// TIA Portal project "MPS_4S_V13_SP1" (V13)

(* hardware
DEVICE "S7300/ET200M-Station_1"  S7-300 station
   slot 0: "Profilschiene_0"  Rail  6ES7 390-1***0-0AA0
   slot 1: "PS 307 5A_1"  PS 307 5A  6ES7 307-1EA00-0AA0
   slot 2: "S7-300 PLC"  CPU 314C-2 PN/DP  6ES7 314-6EH04-0AB0  V3.3
      slot 2: "PROFINET-Schnittstelle_1"  PN-IO
         slot 1: "Port_1"  Port
         slot 2: "Port_2"  Port
      slot 5: "DI 24/DO 16_1"  DI24/DO16
      slot 6: "AI 5/AO 2_1"  AI5/AO2
      slot 7: "Zählen_1"  Counter
      slot 8: "Positionieren_1"  Positioning
   slot 4: "CP 343-2_1"  CP 343-2  6GK7 343-2AH01-0XA0  V3.1
DEVICE "MPS Verteilen"  ET 200S station
   slot 0: "Baugruppenträger_0"  Rail
   slot 0: "Verteilen"  IM 151-1 Standard  6ES7 151-1AA04-0AB0
   slot 1: "PM-E DC24V_1"  PM-E 24VDC  6ES7 138-4CA01-0AA0
   slot 2: "4DI x DC24V ST_1"  4DI x 24VDC ST  6ES7 131-4BD01-0AA0
   slot 3: "4DI x DC24V ST_2"  4DI x 24VDC ST  6ES7 131-4BD01-0AA0
   slot 4: "4DO x DC24V / 0,5A ST_1"  4DO x 24VDC / 0.5A ST  6ES7 132-4BD02-0AA0
   slot 5: "4DO x DC24V / 0,5A ST_2"  4DO x 24VDC / 0.5A ST  6ES7 132-4BD02-0AA0
   slot 6: "4DI x DC24V ST_3"  4DI x 24VDC ST  6ES7 131-4BD01-0AA0
   slot 7: "4DO x DC24V / 0,5A ST_3"  4DO x 24VDC / 0.5A ST  6ES7 132-4BD02-0AA0
   slot 8: "4DO x DC24V / 0,5A ST_4"  4DO x 24VDC / 0.5A ST  6ES7 132-4BD02-0AA0
DEVICE "MPS Pick and Place"  ET 200S station
   slot 0: "Baugruppenträger_0"  Rail
   slot 0: "Pick and Place"  IM 151-1 Standard  6ES7 151-1AA04-0AB0
   slot 1: "PM-E DC24V_1"  PM-E 24VDC  6ES7 138-4CA01-0AA0
   slot 2: "4DI x DC24V ST_1"  4DI x 24VDC ST  6ES7 131-4BD01-0AA0
   slot 3: "4DI x DC24V ST_2"  4DI x 24VDC ST  6ES7 131-4BD01-0AA0
   slot 4: "4DO x DC24V / 0,5A ST_1"  4DO x 24VDC / 0.5A ST  6ES7 132-4BD02-0AA0
   slot 5: "4DO x DC24V / 0,5A ST_2"  4DO x 24VDC / 0.5A ST  6ES7 132-4BD02-0AA0
   slot 6: "4DI x DC24V ST_3"  4DI x 24VDC ST  6ES7 131-4BD01-0AA0
DEVICE "MPS Pressen"  ET 200S station
   slot 0: "Baugruppenträger_0"  Rail
   slot 0: "Pressen"  IM 151-1 Standard  6ES7 151-1AA04-0AB0
   slot 1: "PM-E DC24V_1"  PM-E 24VDC  6ES7 138-4CA01-0AA0
   slot 2: "4DI x DC24V ST_1"  4DI x 24VDC ST  6ES7 131-4BD01-0AA0
   slot 3: "4DI x DC24V ST_2"  4DI x 24VDC ST  6ES7 131-4BD01-0AA0
   slot 4: "4DO x DC24V / 0,5A ST_1"  4DO x 24VDC / 0.5A ST  6ES7 132-4BD02-0AA0
   slot 5: "4DO x DC24V / 0,5A ST_2"  4DO x 24VDC / 0.5A ST  6ES7 132-4BD02-0AA0
   slot 6: "2AI x U ST_1"  2AI x U ST  6ES7 134-4FB01-0AB0
   slot 7: "2AO x U ST_1"  2AO x U ST  6ES7 135-4FB01-0AB0
   slot 8: "4DI x DC24V ST_3"  4DI x 24VDC ST  6ES7 131-4BD01-0AA0
   slot 9: "4DI x DC24V ST_4"  4DI x 24VDC ST  6ES7 131-4BD01-0AA0
   slot 10: "4DO x DC24V / 0,5A ST_3"  4DO x 24VDC / 0.5A ST  6ES7 132-4BD02-0AA0
   slot 11: "4DI x DC24V ST_5"  4DI x 24VDC ST  6ES7 131-4BD01-0AA0
   slot 12: "4DO x DC24V / 0,5A ST_4"  4DO x 24VDC / 0.5A ST  6ES7 132-4BD02-0AA0
*)

// ===== PLC "S7-300 PLC"  CPU 314C-2 PN/DP =====

VAR_GLOBAL   // PLC tag table "Standard-Variablentabelle"
   "Mx_Clock10Hz" AT %M100.0 : Bool;   // CPU-Taktmerker-Bit 0: f=10Hz / T=0.1s
   "Mx_Clock5Hz" AT %M100.1 : Bool;   // CPU-Taktmerker-Bit 1: f=10Hz / T=0.2s
   "Mx_Clock2.5Hz" AT %M100.2 : Bool;   // CPU-Taktmerker-Bit 2: f=10Hz / T=0.4s
   "Mx_Clock2Hz" AT %M100.3 : Bool;   // CPU-Taktmerker-Bit 3: f=10Hz / T=0.5s
   "Mx_Clock1.25Hz" AT %M100.4 : Bool;   // CPU-Taktmerker-Bit 4: f=10Hz / T=0.8s
   "Mx_Clock1Hz" AT %M100.5 : Bool;   // CPU-Taktmerker-Bit 5: f=10Hz / T=1s
   "Mx_Clock0.625Hz" AT %M100.6 : Bool;   // CPU-Taktmerker-Bit 6: f=10Hz / T=1.6s
   "Mx_Clock0.5Hz" AT %M100.7 : Bool;   // CPU-Taktmerker-Bit 7: f=10Hz / T=2s
   "Ix_OnButton" AT %I1.0 : Bool;   // Bedienpult: S1, Starttaster
   "Ix_OffButton" AT %I1.1 : Bool;   // Bedienpult: S2, Stopptaster (NC)
   "Ix_KeySwitch" AT %I1.2 : Bool;   // Bedienpult: S3, Schlüsselschalter
   "Ix_ResetButton" AT %I1.3 : Bool;   // Bedienpult: S4, Resettaster (Richten)
   "Qx_OnSignalLamp" AT %Q1.0 : Bool;   // Bedienpult: P1, Startlampe
   "Qx_ResetSignalLamp" AT %Q1.1 : Bool;   // Bedienpult: P2, Resetlampe (Richten)
   "Qx_EmergencyStopSignalLamp" AT %Q1.2 : Bool;   // Bedienpult: P3, NOT-AUS-Lampe
   "Qx_KeySwitchSignalLamp" AT %Q1.3 : Bool;   // Bedienpult: P4, Schlüsselschalter-Lampe
   "Ix_EmergencyStop" AT %I64.1 : Bool;   // NOT-AUS aktiv
   "Mx_Enable" AT %M10.0 : Bool;   // Schrittfreigabe in der Ablaufkette
   "Mx_OnFlag" AT %M10.1 : Bool;   // Startmerker
   "Mx_InitBit" AT %M10.2 : Bool;   // Initialisierungsbit
   "Qb_Panel" AT %QB1 : Byte;   // Ausgangsbyte Bedienpult
   "Qx_HazardousConditionsSignalTower" AT %Q4.3 : Bool;   // Signalsäule rot: P13, Gefahr, Alarm
   "Qx_NormalConditionsSignalTower" AT %Q4.1 : Bool;   // Signalsäule grün: P11, Normaler, sicherer Betriebszustand
   "Qx_DangerousConditionsImminentSignalTower" AT %Q4.2 : Bool;   // Signalsäule gelb: P12, Vorsicht, abnormaler, kritischer Zustand
   "Qx_NoParticularMeaningSignalTower" AT %Q4.0 : Bool;   // Signalsäule weiss: P10, Neutral, allgemeine Information
   "Mx_PEdgeFlag_Step1" AT %M10.4 : Bool;   // Positiver Flankenmerker für Schritt 1
   "Mx_E-StopStep02" AT %M10.5 : Bool;   // NOT-AUS-Sequenz: Schritt 2
   "Mx_E-StopStep01" AT %M10.3 : Bool;   // NOT-AUS-Sequenz: Schritt 1
END_VAR

VAR_GLOBAL   // PLC tag table "Verteilen_Variablentabelle"
   "Mx_DistrStep10" AT %M30.1 : Bool;   // Station Verteilen: Schritt 10
   "Mx_DistrStep11" AT %M30.2 : Bool;   // Station Verteilen: Schritt 11
   "Mx_DistrStep12" AT %M30.3 : Bool;   // Station Verteilen: Schritt 12
   "Mx_DistrStep13" AT %M30.4 : Bool;   // Station Verteilen: Schritt 13
   "Mx_DistrStep14" AT %M30.5 : Bool;   // Station Verteilen: Schritt 14
   "Mx_DistrStep15" AT %M30.6 : Bool;   // Station Verteilen: Schritt 15
   "Mx_DistrStep16" AT %M30.7 : Bool;   // Station Verteilen: Schritt 16
   "Mx_DistrStep17" AT %M31.0 : Bool;   // Station Verteilen: Schritt 17
   "Mx_DistrStep18" AT %M31.1 : Bool;   // Station Verteilen: Schritt 18
   "Mx_DistrInitPos" AT %M30.0 : Bool;   // Station Verteilen: Grundstellung
   "Ix_DistrMagazineEmpty" AT %I0.6 : Bool;   // Station Verteilen: B4, Sensor Magazin leer
   "Ix_DistrPickAndPlaceReady" AT %I0.7 : Bool;   // Station Verteilen: IP_FI, Folgestation frei
   "Ix_DistrWorkpieceSuckedIn" AT %I0.3 : Bool;   // Station Verteilen: 2B1, Sensor Werkstück angesaugt
   "Ix_DistrSwivelCylinderPositionMagazine" AT %I0.4 : Bool;   // Station Verteilen: 3S1, Sensor Schwenkzylinder in Position Magazin
   "Ix_DistrSwivelCylinderPositionPickAndPlace" AT %I0.5 : Bool;   // Station Verteilen: 3S2, Sensor Schwenkzylinder in Position Folgestation
   "Ix_DistrEjectCylinderPositionRetracted" AT %I0.2 : Bool;   // Station Verteilen: 1B1, Ausschiebezylinder eingefahren
   "Ix_DistrEjectCylinderPositionAdvanced" AT %I0.1 : Bool;   // Station Verteilen: 1B2, Ausschiebezylinder ausgefahren
   "Qx_DistrEjectCylinderEjectWorkpiece" AT %Q0.0 : Bool;   // Station Verteilen: 1M1, Ausschiebezylinder Werkstück ausschieben
   "Qx_DistrVacuumOn" AT %Q0.1 : Bool;   // Station Verteilen: 2M1, Vakuum ein
   "Qx_DistrPushOutPulse" AT %Q0.2 : Bool;   // Station Verteilen: 2M2, Ausstossimpuls
   "Qx_DistrSwivelCylinderMagazine" AT %Q0.3 : Bool;   // Station Verteilen: 3M1, Schwenkzylinder zum Magazin
   "Qx_DistrSwivelCylinderPickAndPlace" AT %Q0.4 : Bool;   // Station Verteilen: 3M2, Schwenkzylinder zur Folgestation
   "Mb_DistrFlagByte30" AT %MB30 : Byte;   // Station Verteilen: Merkerbyte 30
   "Mb_DistrFlagByte31" AT %MB31 : Byte;   // Station Verteilen: Merkerbyte 31
   "Qb_DistrOutputByte0" AT %QB0 : Byte;   // Station Verteilen: Ausgangsbyte 0
   "Mx_DistrStep19" AT %M31.2 : Bool;   // Station Verteilen: Schritt 19
   "Mx_DistrPEdgeFlag_Step2" AT %M31.7 : Bool;   // Positiver Flankenmerker für Schritt 2
END_VAR

VAR_GLOBAL   // PLC tag table "Pick&Place_Variablentabelle"
   "Mx_PAPStep10" AT %M50.1 : Bool;   // Station Pick & Place: Schritt 10
   "Mx_PAPStep11" AT %M50.2 : Bool;   // Station Pick & Place: Schritt 11
   "Mx_PAPStep12" AT %M50.3 : Bool;   // Station Pick & Place: Schritt 12
   "Mx_PAPStep13" AT %M50.4 : Bool;   // Station Pick & Place: Schritt 13
   "Mx_PAPStep14" AT %M50.5 : Bool;   // Station Pick & Place: Schritt 14
   "Mx_PAPStep15" AT %M50.6 : Bool;   // Station Pick & Place: Schritt 15
   "Mx_PAPStep16" AT %M50.7 : Bool;   // Station Pick & Place: Schritt 16
   "Mx_PAPStep17" AT %M51.0 : Bool;   // Station Pick & Place: Schritt 17
   "Mx_PAPStep18" AT %M51.1 : Bool;   // Station Pick & Place: Schritt 18
   "Mx_PAPStep19" AT %M51.2 : Bool;   // Station Pick & Place: Schritt 19
   "Mx_PAPStep20" AT %M51.3 : Bool;   // Station Pick & Place: Schritt 20
   "Mx_PAPStep21" AT %M51.4 : Bool;   // Station Pick & Place: Schritt 21
   "Mx_PAPStep22" AT %M51.5 : Bool;   // Station Pick & Place: Schritt 22
   "Mx_PAPStep23" AT %M51.6 : Bool;   // Station Pick & Place: Schritt 23
   "Mx_PAPStep24" AT %M51.7 : Bool;   // Station Pick & Place: Schritt 24
   "Mx_PAPStep25" AT %M52.0 : Bool;   // Station Pick & Place: Schritt 25
   "Ix_PAPPartAvailable" AT %I2.0 : Bool;   // Station Pick & Place: PART_AV, Werkstück am Eingang
   "Ix_PAPMiniSlideRetracted" AT %I2.1 : Bool;   // Station Pick & Place: 1B1, Mini-Schlitten eingefahren
   "Ix_PAPMiniSlideAdvanced" AT %I2.2 : Bool;   // Station Pick & Place: 1B2, Mini-Schlitten ausgefahren
   "Ix_PAPMiniSlideOnTop" AT %I2.3 : Bool;   // Station Pick & Place: 2B1, Mini-Schlitten ist oben
   "Ix_PAPMiniSlideDown" AT %I2.4 : Bool;   // Station Pick & Place: 3B1, Mini-Schlitten ist unten
   "Ix_PAPWorkpiecePosB" AT %I2.5 : Bool;   // Station Pick & Place: B1, Werkstück Position B
   "Ix_PAPWorkpiecePosC" AT %I2.6 : Bool;   // Station Pick & Place: B2, Werkstück Position C
   "Ix_PAPPressReady" AT %I2.7 : Bool;   // Station Pick & Place: IP_FI, Folgestation frei
   "Qx_PAPConveyorBeltOn" AT %Q2.0 : Bool;   // Station Pick & Place: M1, Bandmotor ein
   "Qx_PAPMiniSlideMoveOut" AT %Q2.2 : Bool;   // Station Pick & Place: 1M2, Mini-Schlitten ausfahren
   "Qx_PAPMiniSlideMoveDown" AT %Q2.3 : Bool;   // Station Pick & Place: 2M1, Mini-Schlitten nach unten
   "Qx_PAPVacuumOn" AT %Q2.4 : Bool;   // Station Pick & Place: 3M1, Vakuum ein
   "Qx_PAPFeedSeparatorMoveOut" AT %Q2.5 : Bool;   // Station Pick & Place: 4M1, Vereinzeler ausfahren
   "Qx_PAPBusy" AT %Q2.7 : Bool;   // Station Pick & Place: IP_N_FO, Station belegt
   "Mb_PAPFlagByte50" AT %MB50 : Byte;   // Station Pick & Place: Merkerbyte 50
   "Mb_PAPFlagByte51" AT %MB51 : Byte;   // Station Pick & Place: Merkerbyte 51
   "Mb_PAPFlagByte52" AT %MB52 : Byte;   // Station Pick & Place: Merkerbyte 52
   "Qb_PAPOutputByte2" AT %QB2 : Byte;   // Station Pick & Place: Ausgangsbyte 2
   "Mx_PAPInitPos" AT %M50.0 : Bool;   // Station Pick & Place: Grundstellung
   "Ix_PAPWorkpieceInSlide" AT %I4.0 : Bool;   // Station Pick & Place: B3, Werkstückeinsatz in Rutsche
   "Mx_PAPStep26" AT %M52.1 : Bool;   // Station Pick & Place: Schritt 26
   "Mx_PAPPEdgeFlag_Step2" AT %M52.7 : Bool;   // Positiver Flankenmerker für Schritt 2
END_VAR

VAR_GLOBAL   // PLC tag table "Pressen_Variablentabelle"
   "Mx_PressStep10" AT %M70.1 : Bool;   // Station Pressen: Schritt 10
   "Mx_PressStep11a" AT %M70.2 : Bool;   // Station Pressen: Schritt 11a
   "Mx_PressStep11b" AT %M70.3 : Bool;   // Station Pressen: Schritt 11b
   "Mx_PressStep12" AT %M70.4 : Bool;   // Station Pressen: Schritt 12
   "Mx_PressStep13" AT %M70.5 : Bool;   // Station Pressen: Schritt 13
   "Mx_PressStep14" AT %M70.6 : Bool;   // Station Pressen: Schritt 14
   "Mx_PressStep15" AT %M70.7 : Bool;   // Station Pressen: Schritt 15
   "Mx_PressStep16" AT %M71.0 : Bool;   // Station Pressen: Schritt 16
   "Mx_PressStep17" AT %M71.1 : Bool;   // Station Pressen: Schritt 17
   "Mx_PressStep18" AT %M71.2 : Bool;   // Station Pressen: Schritt 18
   "Mx_PressStep19" AT %M71.3 : Bool;   // Station Pressen: Schritt 19
   "Mx_PressStep20" AT %M71.4 : Bool;   // Station Pressen: Schritt 20
   "Mx_PressStep21" AT %M71.5 : Bool;   // Station Pressen: Schritt 21
   "Mx_PressStep22" AT %M71.6 : Bool;   // Station Pressen: Schritt 22
   "Mx_PressStep23" AT %M71.7 : Bool;   // Station Pressen: Schritt 23
   "Ix_PressPartAvailable" AT %I3.0 : Bool;   // Station Pressen: PART_AV, Werkstück im Greifer
   "Ix_PressLinearDrivePositionPickAndPlace" AT %I3.1 : Bool;   // Station Pressen: 2B1, Linearantrieb bei Vorgängerstation
   "Ix_PressLinearDrivePositionRobot" AT %I3.2 : Bool;   // Station Pressen: 2B2, Linearantrieb bei Folgestation
   "Ix_PressRotaryDrivePositionPickAndPlace" AT %I3.3 : Bool;   // Station Pressen: 3B1, Drehantrieb bei Vorgängerstation
   "Ix_PressRotaryDrivePositionProcessing" AT %I3.4 : Bool;   // Station Pressen: 3B2, Drehantrieb bei Bearbeitungsstation
   "Ix_PressRotaryDrivePositionRobot" AT %I3.5 : Bool;   // Station Pressen: 3B3, Drehantrieb bei Folgestation
   "Ix_PressPressureReached" AT %I3.6 : Bool;   // Station Pressen: 4B1, Einpressdruck erreicht
   "Ix_PressRobotReady" AT %I3.7 : Bool;   // Station Pressen: ÏP_FI, Folgestation frei
   "Qx_PressCloseGripper" AT %Q3.0 : Bool;   // Station Pressen: 1M1, Greifer schliessen
   "Qx_PressLinearDriveRobot" AT %Q3.2 : Bool;   // Station Pressen: 2M2, Linearantrieb zur Folgestation
   "Qx_PressRotaryDrivePickAndPlace" AT %Q3.3 : Bool;   // Station Pressen: 3M1, Drehantrieb zur Vorgängerstation
   "Qx_PressRotaryDriveProcessing" AT %Q3.4 : Bool;   // Station Pressen: 3M2, Drehantrieb zur Bearbeitungsstation
   "Qx_PressRotaryDriveRobot" AT %Q3.5 : Bool;   // Station Pressen: 3M3, Drehantrieb zur Folgestation
   "Qx_PressMusclePressurize" AT %Q3.6 : Bool;   // Station Pressen: 4M1, Fluidic Muscle belüften
   "Qx_PressBusy" AT %Q3.7 : Bool;   // Station Pressen: IP_N_FO, Station belegt
   "Mb_PressFlagByte70" AT %MB70 : Byte;   // Station Pressen: Merkerbyte 70
   "Mb_PressFlagByte71" AT %MB71 : Byte;   // Station Pressen: Merkerbyte 71
   "Mb_PressFlagByte72" AT %MB72 : Byte;   // Station Pressen: Merkerbyte 72
   "Mx_PressInitPos" AT %M70.0 : Bool;   // Station Pressen: Grundstellung
   "Qb_PressOutputByte3" AT %QB3 : Byte;   // Station Pressen: Ausgangsbyte 3
   "Iw_PressActualPressureValue" AT %IW66 : Int;   // Station Pressen: Istwert Pressdruck
   "Iw_PressActualPressureValue_4B1" AT %IW68 : Int;   // Station Pressen: Istwert Pressdruck (4B1)
   "Qw_PressSetPressureValue" AT %QW66 : Int;   // Station Pressen: Sollwert Pressdruck
   "Mx_PressStep24" AT %M72.0 : Bool;   // Station Pressen: Schritt 24
   "Mx_PressPEdgeFlag_Step2" AT %M72.7 : Bool;   // Positiver Flankenmerker für Schritt 2
END_VAR

FUNCTION "1a_NOT-STOP_Schrittkette" : Void   // FC1, FBD
TITLE = NOT-STOP-Funktion
{ S7_Optimized_Access := 'FALSE' }
VERSION : 0.1
   VAR_TEMP   // added for the SCL form of the ladder/FBD networks
      _w1 : Bool;
   END_VAR
BEGIN

REGION Network 1: Schritt 1
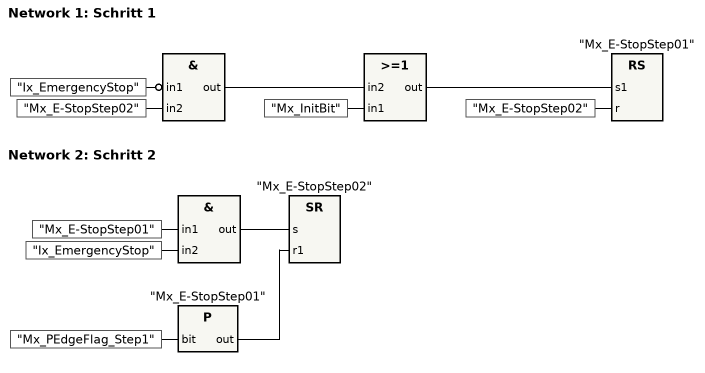
   IF "Mx_E-StopStep02" THEN
       "Mx_E-StopStep01" := FALSE;   // RS flip-flop
   END_IF;
   IF (NOT "Ix_EmergencyStop" AND "Mx_E-StopStep02") OR "Mx_InitBit" THEN "Mx_E-StopStep01" := TRUE; END_IF;
END_REGION

REGION Network 2: Schritt 2
   #_w1 := "Mx_E-StopStep01" AND NOT "Mx_PEdgeFlag_Step1";   // rising edge of "Mx_E-StopStep01"
   "Mx_PEdgeFlag_Step1" := "Mx_E-StopStep01";
   IF "Mx_E-StopStep01" AND "Ix_EmergencyStop" THEN
       "Mx_E-StopStep02" := TRUE;   // SR flip-flop
   END_IF;
   IF #_w1 THEN "Mx_E-StopStep02" := FALSE; END_IF;
END_REGION
END_FUNCTION

FUNCTION "1b_NOT-STOP_Aktionen" : Void   // FC2, FBD
TITLE = Aktionen-Funktion NOT-STOP
{ S7_Optimized_Access := 'FALSE' }
VERSION : 0.1
BEGIN

REGION Network 1: Rücksetzen der Merker der Station VERTEILEN
   // Alle Merker werden zurückgesetzt (der Wert 0 wird in das Merkerbyte "Mb_DistrFlagByte30" geschrieben)
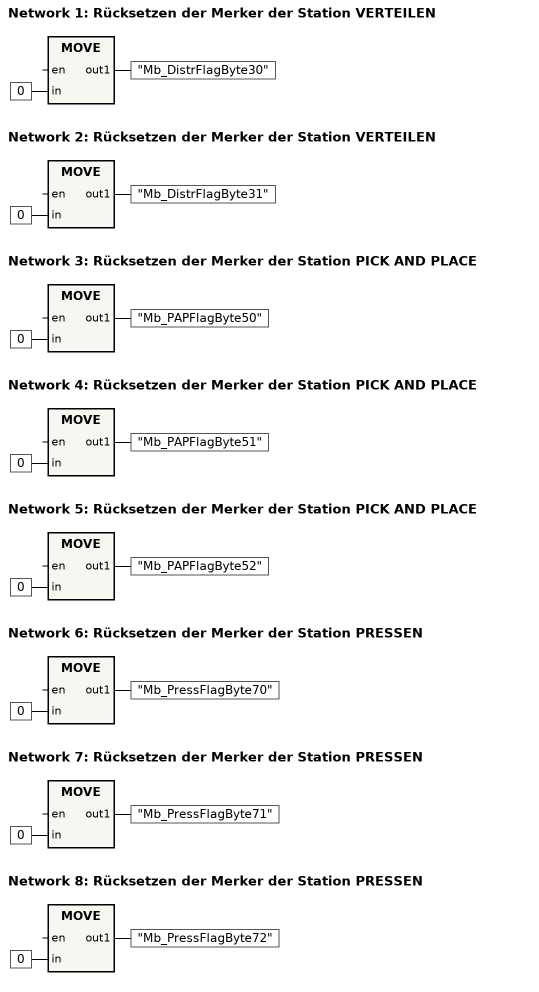
   "Mb_DistrFlagByte30" := 0;
END_REGION

REGION Network 2: Rücksetzen der Merker der Station VERTEILEN
   // Alle Merker werden zurückgesetzt (der Wert 0 wird in das Merkerbyte "Mb_DistrFlagByte31" geschrieben)
   "Mb_DistrFlagByte31" := 0;
END_REGION

REGION Network 3: Rücksetzen der Merker der Station PICK AND PLACE
   // Alle Merker werden zurückgesetzt (der Wert 0 wird in das Merkerbyte "Mb_PAPFlagByte50" geschrieben)
   "Mb_PAPFlagByte50" := 0;
END_REGION

REGION Network 4: Rücksetzen der Merker der Station PICK AND PLACE
   // Alle Merker werden zurückgesetzt (der Wert 0 wird in das Merkerbyte "Mb_PAPFlagByte51" geschrieben)
   "Mb_PAPFlagByte51" := 0;
END_REGION

REGION Network 5: Rücksetzen der Merker der Station PICK AND PLACE
   // Alle Merker werden zurückgesetzt (der Wert 0 wird in das Merkerbyte "Mb_PAPFlagByte52" geschrieben)
   "Mb_PAPFlagByte52" := 0;
END_REGION

REGION Network 6: Rücksetzen der Merker der Station PRESSEN
   // Alle Merker werden zurückgesetzt (der Wert 0 wird in das Merkerbyte "Mb_PressFlagByte70" geschrieben)
   "Mb_PressFlagByte70" := 0;
END_REGION

REGION Network 7: Rücksetzen der Merker der Station PRESSEN
   // Alle Merker werden zurückgesetzt (der Wert 0 wird in das Merkerbyte "Mb_PressFlagByte71" geschrieben)
   "Mb_PressFlagByte71" := 0;
END_REGION

REGION Network 8: Rücksetzen der Merker der Station PRESSEN
   // Alle Merker werden zurückgesetzt (der Wert 0 wird in das Merkerbyte "Mb_PressFlagByte72" geschrieben)
   "Mb_PressFlagByte72" := 0;
END_REGION
END_FUNCTION

FUNCTION "2_MPS_Grundstellung" : Void   // FC3, FBD
TITLE = Grundstellung MPS
{ S7_Optimized_Access := 'FALSE' }
VERSION : 0.1
BEGIN

REGION Network 1: Grundstellung Station VERTEILEN abfragen
   // Die Station Verteilen ist in der Grundstellung, wenn der Ausschiebezylinder ausgefahren ist, der Schwenkzylinder sich bei der Position Folgestation befindet, und das Vakuum ausgeschaltet ist.
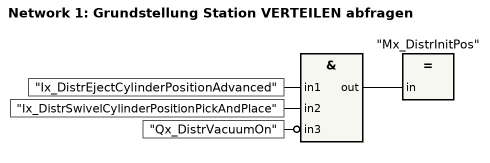
   "Mx_DistrInitPos" := "Ix_DistrEjectCylinderPositionAdvanced" AND "Ix_DistrSwivelCylinderPositionPickAndPlace" AND NOT "Qx_DistrVacuumOn";
END_REGION

REGION Network 2: Grundstellung Station PICK AND PLACE abfragen
END_REGION

REGION Network 3: Grundstellung Station PRESSEN abfragen
END_REGION
END_FUNCTION

FUNCTION "3_Signalisierung_Aktionen" : Void   // FC4, FBD
TITLE = Signalisierung
{ S7_Optimized_Access := 'FALSE' }
VERSION : 0.1
// WICHTIG: Jeder Aktor (Ausgang) darf nur einmal in der Befehlsausgabe angesteuert werden. Falls ein Aktor in verschiedenen Schritten aktiv ist, werden ihm die jeweiligen Schrittmerker über eine ODER-Verknüpfung zugewiesen.
BEGIN

REGION Network 1: NOT-.AUS-Lampe
   // WICHTIG: In der Hardwarekonfiguration muss das Taktmerkerbyte 100 aktiviert werden. Die Hardware muss in die CPU geladen werden.
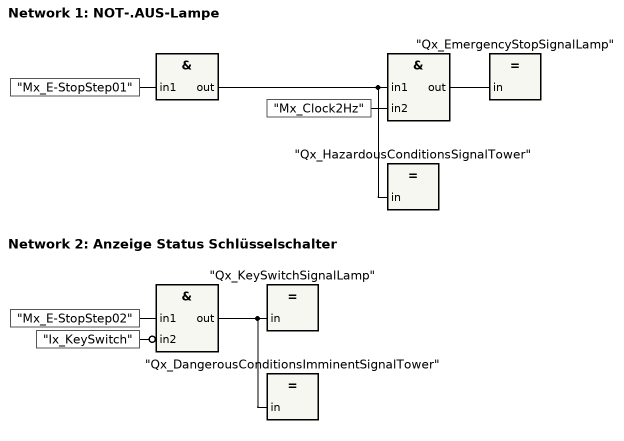
   "Qx_EmergencyStopSignalLamp" := "Mx_E-StopStep01" AND "Mx_Clock2Hz";
   "Qx_HazardousConditionsSignalTower" := "Mx_E-StopStep01";
END_REGION

REGION Network 2: Anzeige Status Schlüsselschalter
   // Bei Betätigung des Schlüsselschalters bleibt die Anlage im jeweils aktuellen Schritt stehen. Die Meldelampe leuchtet.
   "Qx_KeySwitchSignalLamp" := "Mx_E-StopStep02" AND NOT "Ix_KeySwitch";
   "Qx_DangerousConditionsImminentSignalTower" := "Qx_KeySwitchSignalLamp";
END_REGION

REGION Network 3: Anzeige Grundstellung (Reset)
END_REGION

REGION Network 4: Anzeige Starttaste verlangt
   // WICHTIG: In der Hardwarekonfiguration muss das Taktmerkerbyte 100 aktiviert werden. Die Hardware muss in die CPU geladen werden.
END_REGION
END_FUNCTION

FUNCTION "4a_Verteilen_Schrittkette" : Void   // FC30, FBD
TITLE = Schrittkette Station Verteilen
{ S7_Optimized_Access := 'FALSE' }
VERSION : 0.1
   VAR_TEMP   // added for the SCL form of the ladder/FBD networks
      _w1 : Bool;
   END_VAR
BEGIN

REGION Network 1: Schritt 10
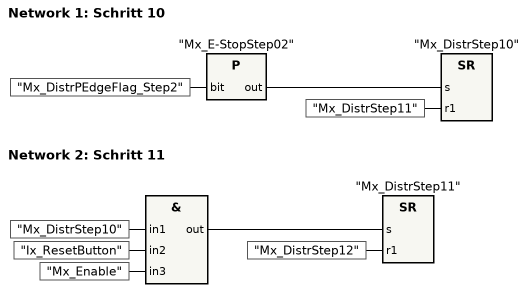
   #_w1 := "Mx_E-StopStep02" AND NOT "Mx_DistrPEdgeFlag_Step2";   // rising edge of "Mx_E-StopStep02"
   "Mx_DistrPEdgeFlag_Step2" := "Mx_E-StopStep02";
   IF #_w1 THEN
       "Mx_DistrStep10" := TRUE;   // SR flip-flop
   END_IF;
   IF "Mx_DistrStep11" THEN "Mx_DistrStep10" := FALSE; END_IF;
END_REGION

REGION Network 2: Schritt 11
   IF "Mx_DistrStep10" AND "Ix_ResetButton" AND "Mx_Enable" THEN
       "Mx_DistrStep11" := TRUE;   // SR flip-flop
   END_IF;
   IF "Mx_DistrStep12" THEN "Mx_DistrStep11" := FALSE; END_IF;
END_REGION

REGION Network 3: Schritt 12
END_REGION

REGION Network 4: Schritt 13
END_REGION

REGION Network 5: Schritt 14
END_REGION

REGION Network 6: Schritt 15
END_REGION

REGION Network 7: Schritt 16
END_REGION

REGION Network 8: Schritt 17
END_REGION

REGION Network 9: Schritt 18
END_REGION

REGION Network 10: Schritt 19
END_REGION
END_FUNCTION

FUNCTION "4b_Verteilen_Aktionen" : Void   // FC31, FBD
TITLE = Befehlsausgabe Station Verteilen
{ S7_Optimized_Access := 'FALSE' }
VERSION : 0.1
// WICHTIG: Jeder Aktor (Ausgang) darf nur einmal in der Befehlsausgabe angesteuert werden. Falls ein Aktor in verschiedenen Schritten aktiv ist, werden ihm die jeweiligen Schrittmerker über eine ODER-Verknüpfung zugewiesen.
BEGIN

REGION Network 1: Schwenkzylinder zur Position Magazin
END_REGION

REGION Network 2: Schwenkzylinder zur Position Pick And Place
END_REGION

REGION Network 3: Ausschiebezylinder
END_REGION

REGION Network 4: Vakuum
END_REGION

REGION Network 5: Ausstossimpuls
END_REGION
END_FUNCTION

FUNCTION "5a_PickAndPlace_Schrittkette" : Void   // FC50, FBD
{ S7_Optimized_Access := 'FALSE' }
VERSION : 0.1
BEGIN
END_FUNCTION

FUNCTION "5b_PickAndPlace_Aktionen" : Void   // FC51, FBD
{ S7_Optimized_Access := 'FALSE' }
VERSION : 0.1
BEGIN
END_FUNCTION

FUNCTION "6a_Pressen_Schrittkette" : Void   // FC70, FBD
{ S7_Optimized_Access := 'FALSE' }
VERSION : 0.1
BEGIN
END_FUNCTION

FUNCTION "6b_Pressen_Aktionen" : Void   // FC71, FBD
{ S7_Optimized_Access := 'FALSE' }
VERSION : 0.1
BEGIN
END_FUNCTION

ORGANIZATION_BLOCK "0b_Main"   // OB1, FBD
TITLE = Hauptbaustein / "Main Program Sweep (Cycle)"
{ S7_Optimized_Access := 'FALSE' }
VERSION : 0.1
BEGIN

REGION Network 1: Aufruf Schrittkette-Funktion NOT-STOP (E-Stop main sequence)
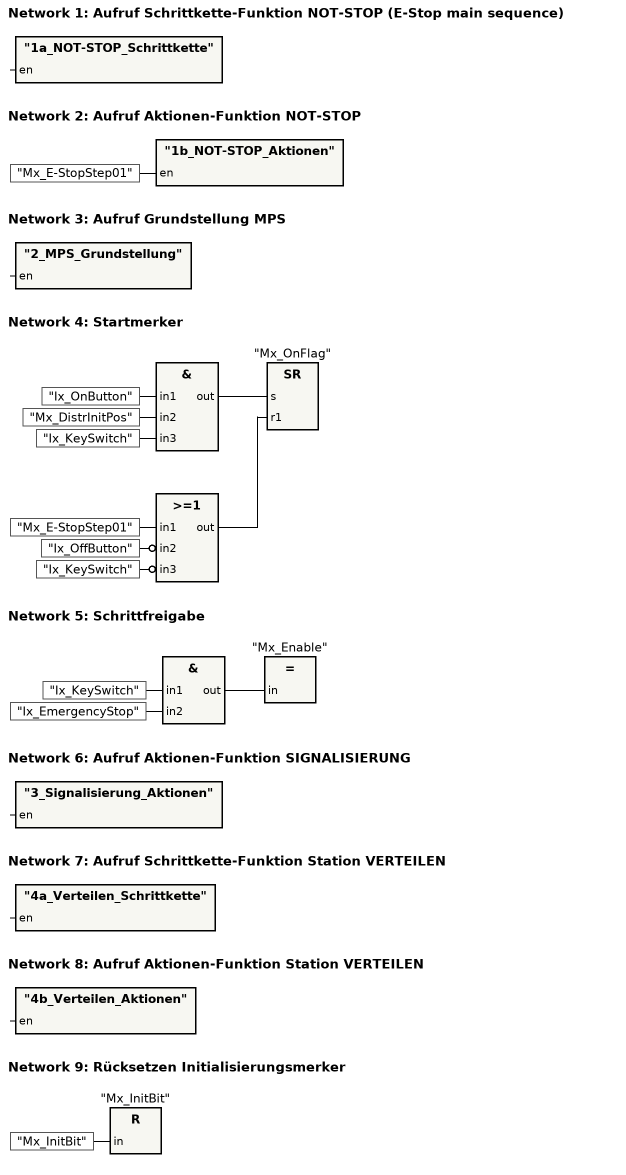
   "1a_NOT-STOP_Schrittkette"();
END_REGION

REGION Network 2: Aufruf Aktionen-Funktion NOT-STOP
   IF "Mx_E-StopStep01" THEN "1b_NOT-STOP_Aktionen"(); END_IF;
END_REGION

REGION Network 3: Aufruf Grundstellung MPS
   "2_MPS_Grundstellung"();
END_REGION

REGION Network 4: Startmerker
   // Der Merker "Mx_OnFlag"wird gesetzt, wenn in der Grundstellung der Anlage(n) der Starttaster betätigt wird und der Schlüsselschalter auf "manuell" steht. Der Merker "Mx_OnFlag" wird in der Schlüsselschalterstellung "manuell" oder wenn NOT-STOP aktiv ist oder wenn der Stopptaster betätigt wird , zurückgesetzt.
   IF "Ix_OnButton" AND "Mx_DistrInitPos" AND "Ix_KeySwitch" THEN
       "Mx_OnFlag" := TRUE;   // SR flip-flop
   END_IF;
   IF "Mx_E-StopStep01" OR NOT "Ix_OffButton" OR NOT "Ix_KeySwitch" THEN "Mx_OnFlag" := FALSE; END_IF;
END_REGION

REGION Network 5: Schrittfreigabe
   // Bei Betätigung des Schlüsselschalters bleibt die Anlage im jeweils aktuellen Schritt stehen.
   "Mx_Enable" := "Ix_KeySwitch" AND "Ix_EmergencyStop";
END_REGION

REGION Network 6: Aufruf Aktionen-Funktion SIGNALISIERUNG
   // WICHTIG: Jeder Aktor (Ausgang) darf nur einmal in der Befehlsausgabe angesteuert werden. Falls ein Aktor in verschiedenen Schritten aktiv ist, werden ihm die jeweiligen Schrittmerker über eine ODER-Verknüpfung zugewiesen.
   "3_Signalisierung_Aktionen"();
END_REGION

REGION Network 7: Aufruf Schrittkette-Funktion Station VERTEILEN
   // Die Schrittkette-Funktion wird zyklisch bearbeitet. Die Merker der Schrittkette werden beim Einschalten der SPS im OB100 oder wenn NOT-STOP aktiv ist im FC2 initialisiert. Mit dem Initialisieren werden alle Schrittmerker zurückgesetzt (mit "0" überschrieben.
   "4a_Verteilen_Schrittkette"();
END_REGION

REGION Network 8: Aufruf Aktionen-Funktion Station VERTEILEN
   // WICHTIG: Jeder Aktor (Ausgang) darf nur einmal in der Befehlsausgabe angesteuert werden. Falls ein Aktor in verschiedenen Schritten aktiv ist, werden ihm die jeweiligen Schrittmerker über eine ODER-Verknüpfung zugewiesen.
   "4b_Verteilen_Aktionen"();
END_REGION

REGION Network 9: Rücksetzen Initialisierungsmerker
   // Der Initialiserungsmerker "Mx_InitBit" wird beim Übergang STOP nach RUN der CPU im OB100 gesetzt und nach dem ersten Programmzyklus im letzten (!) Netzwerk des OB1 wieder zurückgesetzt.
   IF "Mx_InitBit" THEN "Mx_InitBit" := FALSE; END_IF;
END_REGION
END_ORGANIZATION_BLOCK

ORGANIZATION_BLOCK "0a_Anlaufbaustein"   // OB100, FBD
TITLE = Anlaufbaustein / "Complete Restart"
{ S7_Optimized_Access := 'FALSE' }
VERSION : 0.1
// Der Anlaufbaustein (Complete Restart) wird beim Übergang STOP nach RUN der CPU im allerersten Programmzyklus ein einziges Mal durchlaufen. Der Anlaufbaustein setzt alle Merker und Ausgänge der Station(en) zurück. Der Initialisierungsmerker "Mx_InitBit" wird als einziger Merker gesetzt. Dieser Merker soll für einen Zyklus 1-Signal haben und im letzten Netzwerk von OB1 wieder zurückgesetzt werden.
BEGIN

REGION Network 1: Rücksetzen der Bedienpultausgänge
   // Alle Ausgänge des Bedienpults (Signallampen) werden zurückgesetzt (der Wert 0 wird in das Ausgangsbyte QB1 geschrieben.
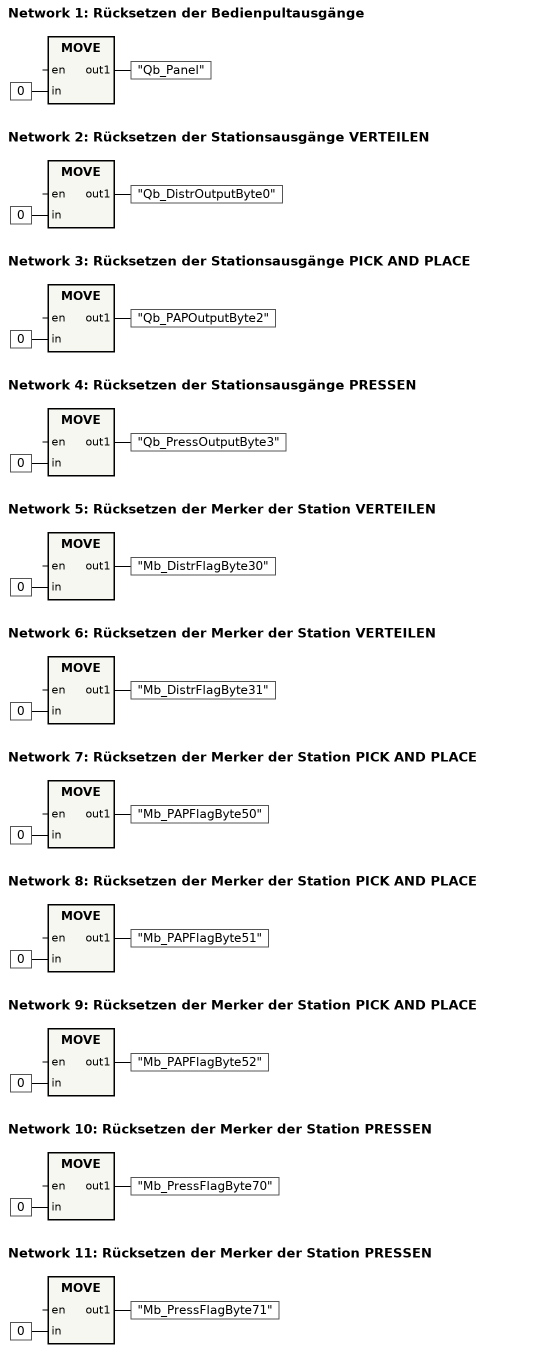
   "Qb_Panel" := 0;
END_REGION

REGION Network 2: Rücksetzen der Stationsausgänge VERTEILEN
   // Alle Ausgänge der Station werden zurückgesetzt (der Wert 0 wird in das Ausgangsbyte QB0 geschrieben.
   "Qb_DistrOutputByte0" := 0;
END_REGION

REGION Network 3: Rücksetzen der Stationsausgänge PICK AND PLACE
   // Alle Ausgänge der Station werden zurückgesetzt (der Wert 0 wird in das Ausgangsbyte QB2 geschrieben.
   "Qb_PAPOutputByte2" := 0;
END_REGION

REGION Network 4: Rücksetzen der Stationsausgänge PRESSEN
   // Alle Ausgänge der Station werden zurückgesetzt (der Wert 0 wird in das Ausgangsbyte QB3 geschrieben.
   "Qb_PressOutputByte3" := 0;
END_REGION

REGION Network 5: Rücksetzen der Merker der Station VERTEILEN
   // Alle Merker werden zurückgesetzt (der Wert 0 wird in das Merkerbyte "Mb_DistrFlagByte30" geschrieben)
   "Mb_DistrFlagByte30" := 0;
END_REGION

REGION Network 6: Rücksetzen der Merker der Station VERTEILEN
   // Alle Merker werden zurückgesetzt (der Wert 0 wird in das Merkerbyte "Mb_DistrFlagByte31" geschrieben)
   "Mb_DistrFlagByte31" := 0;
END_REGION

REGION Network 7: Rücksetzen der Merker der Station PICK AND PLACE
   // Alle Merker werden zurückgesetzt (der Wert 0 wird in das Merkerbyte "Mb_PAPFlagByte50" geschrieben)
   "Mb_PAPFlagByte50" := 0;
END_REGION

REGION Network 8: Rücksetzen der Merker der Station PICK AND PLACE
   // Alle Merker werden zurückgesetzt (der Wert 0 wird in das Merkerbyte "Mb_PAPFlagByte51" geschrieben)
   "Mb_PAPFlagByte51" := 0;
END_REGION

REGION Network 9: Rücksetzen der Merker der Station PICK AND PLACE
   // Alle Merker werden zurückgesetzt (der Wert 0 wird in das Merkerbyte "Mb_PAPFlagByte52" geschrieben)
   "Mb_PAPFlagByte52" := 0;
END_REGION

REGION Network 10: Rücksetzen der Merker der Station PRESSEN
   // Alle Merker werden zurückgesetzt (der Wert 0 wird in das Merkerbyte "Mb_PressFlagByte70" geschrieben)
   "Mb_PressFlagByte70" := 0;
END_REGION

REGION Network 11: Rücksetzen der Merker der Station PRESSEN
   // Alle Merker werden zurückgesetzt (der Wert 0 wird in das Merkerbyte "Mb_PressFlagByte71" geschrieben)
   "Mb_PressFlagByte71" := 0;
END_REGION

REGION Network 12: Rücksetzen der Merker der Station PRESSEN
   // Alle Merker werden zurückgesetzt (der Wert 0 wird in das Merkerbyte "Mb_PressFlagByte72" geschrieben)
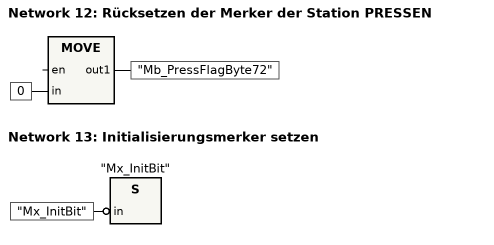
   "Mb_PressFlagByte72" := 0;
END_REGION

REGION Network 13: Initialisierungsmerker setzen
   // Der Initialisierungsmerker "Mx_InitBit" wird gesetzt.
   IF NOT "Mx_InitBit" THEN "Mx_InitBit" := TRUE; END_IF;
END_REGION
END_ORGANIZATION_BLOCK